// TIA Portal V18 export
DATA_BLOCK "State"   // DB3
VERSION : 0.1
// stored: Access Published, AutoNumber true, DBAccessibleFromOPCUA true, DBAccessibleFromWebserver true, IsOnlyStoredInLoadMemory false, IsRetainMemResEnabled false, IsWriteProtectedInAS false, MemoryReserve 100, Namespace Coagulation
   VAR
      Process_done : Bool;
   END_VAR
BEGIN
END_DATA_BLOCK
